TYPE U_APP_INFO :
UNION
  stState             : ST_APP_INFO;
  byState   AT %Q*    : ARRAY[1..SIZEOF(ST_APP_INFO)] OF BYTE;
END_UNION
END_TYPE

(* stored: Version 1.1.0.1, ProductVersion 3.1.4026.20
   DUT U_APP_INFO: Id {a8f5f8f9-bd51-4bb0-bfa4-4802eac82f7e} *)
